// TIA Portal project "Fan Speed Control" (V18)
// 4 speed control for industrial fan

(* hardware
DEVICE "S7-1200 station_1"  S7-1200 Station
   slot 0: "Rack_0"  S7-1200 Rack  Rack  V1.0
   slot 1: "PLC_1"  CPU 1212C AC/DC/Rly  6ES7 212-1BE40-0XB0  V4.6
*)

// ===== PLC "PLC_1"  CPU 1212C AC/DC/Rly =====

VAR_GLOBAL   // PLC tag table "I/O"
   "SPEED_UP" AT %I0.0 : Bool;   // PUSHBUTTON SPEED UP
   "SPEED_DOWN" AT %I0.1 : Bool;   // PUSHBUTTON SPEED DOWN
   "STOP_PROCESS" AT %I0.2 : Bool;   // PUSHBUTTON STOP PROCESS
   "EMERGENCY_STOP" AT %I0.3 : Bool;   // EMERGENCY STOP
   "SPEED_1" AT %Q0.0 : Bool;   // SPEED 1
   "SPEED_2" AT %Q0.1 : Bool;   // SPEED 2
   "SPEED_3" AT %Q0.2 : Bool;   // SPEED 3
   "SPEED_4" AT %Q0.3 : Bool;   // SPEED 4
   "SET_PROCESS" AT %M0.0 : Bool;   // SET INITIAL PROCESS
   "M_COUNT_UP" AT %M0.1 : Bool;   // ACTIVATE COUNT UP
   "M_COUNT_DOWN" AT %M0.2 : Bool;   // ACTIVE COUNT DOWN
   "M_RESET_COUNTER" AT %M0.3 : Bool;   // ACTIVE RESET COUNTER
   "ACTIVATED_INCREMENT" AT %M0.4 : Bool;
   "ACTIVATED_DECREMENT" AT %M0.5 : Bool;
END_VAR

// folder: System blocks/Program resources

DATA_BLOCK "TIMER_SPEED_1"   // DB1
{ S7_Optimized_Access := 'TRUE' }
AUTHOR : Simatic
FAMILY : IEC
NAME : IEC_TMR
VERSION : 1.0
// stored: InstanceOfName IEC_TIMER
"IEC_TIMER"
BEGIN
END_DATA_BLOCK

DATA_BLOCK "COUNTER_SPEEDS"   // DB3
{ S7_Optimized_Access := 'TRUE' }
AUTHOR : Simatic
FAMILY : IEC
NAME : CNTR
VERSION : 1.0
// stored: InstanceOfName IEC_COUNTER
"IEC_COUNTER"
BEGIN
END_DATA_BLOCK

DATA_BLOCK "TIMER_SPEED_2"   // DB7
{ S7_Optimized_Access := 'TRUE' }
AUTHOR : Simatic
FAMILY : IEC
NAME : IEC_TMR
VERSION : 1.0
// stored: InstanceOfName IEC_TIMER
"IEC_TIMER"
BEGIN
END_DATA_BLOCK

DATA_BLOCK "TIMER_SPEED_3"   // DB8
{ S7_Optimized_Access := 'TRUE' }
AUTHOR : Simatic
FAMILY : IEC
NAME : IEC_TMR
VERSION : 1.0
// stored: InstanceOfName IEC_TIMER
"IEC_TIMER"
BEGIN
END_DATA_BLOCK

DATA_BLOCK "TIMER_SPEED_4"   // DB9
{ S7_Optimized_Access := 'TRUE' }
AUTHOR : Simatic
FAMILY : IEC
NAME : IEC_TMR
VERSION : 1.0
// stored: InstanceOfName IEC_TIMER
"IEC_TIMER"
BEGIN
END_DATA_BLOCK

// folder: (top level)

FUNCTION "COUNTER_FUNC" : Void   // FC1, LAD
{ S7_Optimized_Access := 'TRUE' }
VERSION : 0.1
BEGIN

REGION Network 1: SET INITIAL PROCESS
   // SET INITIAL PROCESS
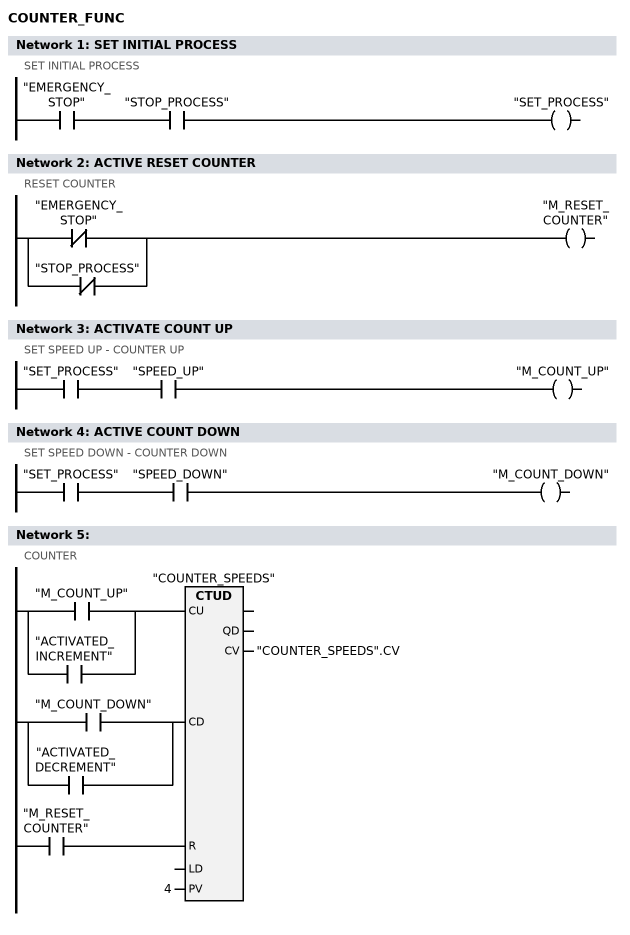
   RUNG wire#powerrail
      Contact( "EMERGENCY_STOP" )
      Contact( "STOP_PROCESS" )
      Coil( "SET_PROCESS" )
   END_RUNG
   // the same network as SCL:
   "SET_PROCESS" := "EMERGENCY_STOP" AND "STOP_PROCESS";
END_REGION

REGION Network 2: ACTIVE RESET COUNTER
   // RESET COUNTER
   RUNG wire#powerrail
      I_Contact( "EMERGENCY_STOP" )
      wire#w1
      Coil( "M_RESET_COUNTER" )
   END_RUNG
   RUNG wire#powerrail
      I_Contact( "STOP_PROCESS" )
   END_RUNG wire#w1
   // the same network as SCL:
   "M_RESET_COUNTER" := NOT "EMERGENCY_STOP" OR NOT "STOP_PROCESS";
END_REGION

REGION Network 3: ACTIVATE COUNT UP
   // SET SPEED UP - COUNTER UP
   RUNG wire#powerrail
      Contact( "SET_PROCESS" )
      Contact( "SPEED_UP" )
      Coil( "M_COUNT_UP" )
   END_RUNG
   // the same network as SCL:
   "M_COUNT_UP" := "SET_PROCESS" AND "SPEED_UP";
END_REGION

REGION Network 4: ACTIVE COUNT DOWN
   // SET SPEED DOWN - COUNTER DOWN
   RUNG wire#powerrail
      Contact( "SET_PROCESS" )
      Contact( "SPEED_DOWN" )
      Coil( "M_COUNT_DOWN" )
   END_RUNG
   // the same network as SCL:
   "M_COUNT_DOWN" := "SET_PROCESS" AND "SPEED_DOWN";
END_REGION

REGION Network 5
   // COUNTER
   "COUNTER_SPEEDS".CTUD(CU := "M_COUNT_UP" OR "ACTIVATED_INCREMENT",
                         CD := "M_COUNT_DOWN" OR "ACTIVATED_DECREMENT",
                         R := "M_RESET_COUNTER",
                         PV := 4,
                         CV => "COUNTER_SPEEDS".CV);
END_REGION
END_FUNCTION

FUNCTION "COUNTER_SPEED_COMPARATOR" : Void   // FC2, LAD
{ S7_Optimized_Access := 'TRUE' }
VERSION : 0.1
BEGIN

REGION Network 1: SPEED 1
   // SPEED 1 - FIRST PULSE
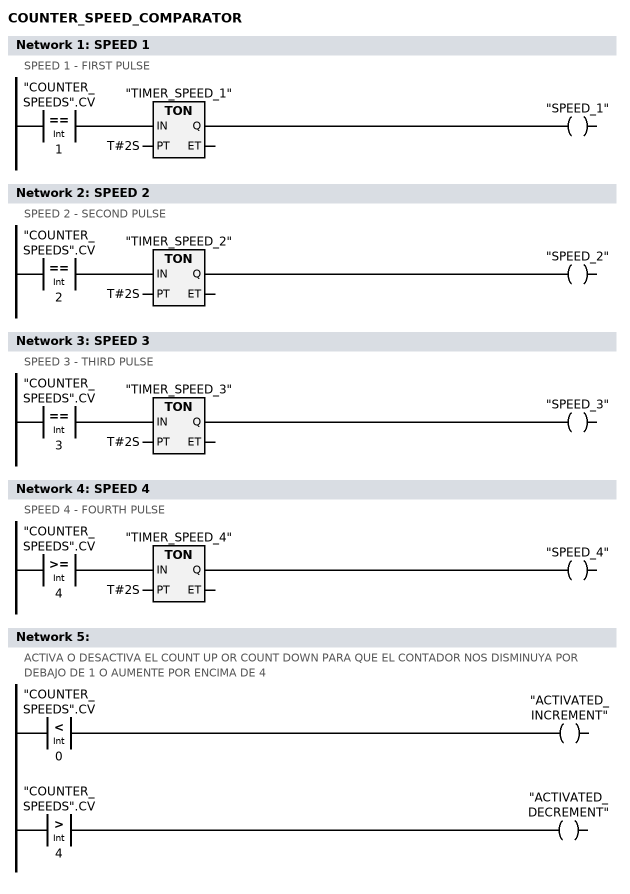
   "TIMER_SPEED_1".TON(IN := "COUNTER_SPEEDS".CV = 1, PT := T#2S);
   "SPEED_1" := "TIMER_SPEED_1".Q;
END_REGION

REGION Network 2: SPEED 2
   // SPEED 2 - SECOND PULSE
   "TIMER_SPEED_2".TON(IN := "COUNTER_SPEEDS".CV = 2, PT := T#2S);
   "SPEED_2" := "TIMER_SPEED_2".Q;
END_REGION

REGION Network 3: SPEED 3
   // SPEED 3 - THIRD PULSE
   "TIMER_SPEED_3".TON(IN := "COUNTER_SPEEDS".CV = 3, PT := T#2S);
   "SPEED_3" := "TIMER_SPEED_3".Q;
END_REGION

REGION Network 4: SPEED 4
   // SPEED 4 - FOURTH PULSE
   "TIMER_SPEED_4".TON(IN := "COUNTER_SPEEDS".CV >= 4, PT := T#2S);
   "SPEED_4" := "TIMER_SPEED_4".Q;
END_REGION

REGION Network 5
   // ACTIVA O DESACTIVA EL COUNT UP OR COUNT DOWN PARA QUE EL CONTADOR NOS DISMINUYA POR DEBAJO DE 1 O AUMENTE POR ENCIMA DE 4
   RUNG wire#powerrail
      { S7_Templates := "SrcType := Int" } LT_Contact(in1 := "COUNTER_SPEEDS".CV, in2 := 0)
      Coil( "ACTIVATED_INCREMENT" )
   END_RUNG
   RUNG wire#powerrail
      { S7_Templates := "SrcType := Int" } GT_Contact(in1 := "COUNTER_SPEEDS".CV, in2 := 4)
      Coil( "ACTIVATED_DECREMENT" )
   END_RUNG
   // the same network as SCL:
   "ACTIVATED_INCREMENT" := "COUNTER_SPEEDS".CV < 0;
   "ACTIVATED_DECREMENT" := "COUNTER_SPEEDS".CV > 4;
END_REGION
END_FUNCTION

ORGANIZATION_BLOCK "Main"   // OB1, LAD, ProgramCycle
TITLE = "Main Program Sweep (Cycle)"
{ S7_Optimized_Access := 'TRUE' }
VERSION : 0.1
   VAR_INPUT
      Initial_Call : Bool;   // Initial call of this OB
      Remanence : Bool;   // =True, if remanent data are available
   END_VAR
BEGIN

REGION Network 1
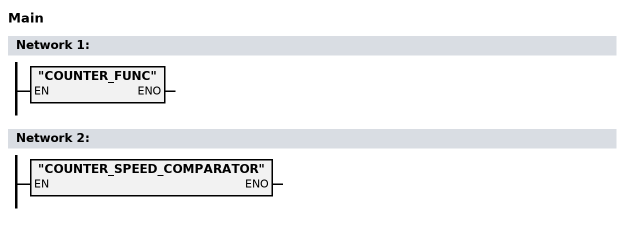
   RUNG wire#powerrail
      "COUNTER_FUNC"()
   END_RUNG
   // the same network as SCL:
   "COUNTER_FUNC"();
END_REGION

REGION Network 2
   RUNG wire#powerrail
      "COUNTER_SPEED_COMPARATOR"()
   END_RUNG
   // the same network as SCL:
   "COUNTER_SPEED_COMPARATOR"();
END_REGION
END_ORGANIZATION_BLOCK